INTERFACE ITF_TopElement1

END_INTERFACE

(* stored: Version 1.1.0.1, ProductVersion 3.1.4024.15
   Itf ITF_TopElement1: Id {34d47d0e-ae89-48cf-972f-3dc3d434f7ac} *)
